(* IEC 61131-3 sources: platform/iec61131/st/osoST/examples, 8 files *)

(* ---- array.st ---- *)
VAR_GLOBAL
  a : ARRAY[0..4] OF DINT;
  i : DINT := 0;
  sum : DINT := 0;
END_VAR

PROCEDURE main()
  FOR i := 0 TO 4 DO
    a[i] := i * 10;
  END_FOR;
  sum := 0;
  FOR i := 0 TO 4 DO
    sum := sum + a[i];
  END_FOR;
  debug(sum);
  debug(a[2]);
END_PROCEDURE

(* ---- array_real.st ---- *)
VAR_GLOBAL
  r : ARRAY[1..3] OF REAL;
  s : REAL := 0.0;
END_VAR

PROCEDURE main()
  r[1] := 1.5;
  r[2] := r[1] * 2.0;
  r[3] := r[2] + r[1];
  s := r[1] + r[2] + r[3];
  debug(s);
  debug(r[3]);
END_PROCEDURE

(* ---- blink.st ---- *)
(* ============================================================
   osoLogic — IEC 61131-3 Structured Text example
   blink.st — LED blink using a counter and trap calls

   Copyright (C) 2026 Angel Miguel Zúñiga Schmemund <miguel@ibercomp.com>
                 Ibercomp SL, Roig Borrell SL

   Part of the osoLogic open-source PLC project — osologic.org
   SPDX-License-Identifier: AGPL-3.0-or-later

   Description / Descripción:
     Toggle a GPIO output every N scan cycles.
     Alterna una salida GPIO cada N ciclos de scan.

   Traps used / Traps utilizados:
     gpio_write(pin, value)  — trap #10
     millis()                — trap #12  (returns I32 milliseconds)
   ============================================================ *)

(* Hardware traps — link to hardware_linux.c or hardware_bare.c
   Traps de hardware — enlazar con hardware_linux.c o hardware_bare.c *)
TRAP gpio_write(pin : DINT; value : DINT) TRAP #10;
TRAP gpio_read(pin : DINT) : DINT        TRAP #11;
TRAP millis() : DINT                     TRAP #12;

(* ── Global state / Estado global ──────────────────────── *)
VAR_GLOBAL
  led_state    : BOOL  := FALSE;
  last_toggle  : DINT  := 0;
END_VAR

(* ── Constants / Constantes ─────────────────────────────── *)
VAR_GLOBAL
  LED_PIN      : DINT  := 0;   (* GPIO pin number / Número de pin GPIO *)
  BLINK_MS     : DINT  := 500; (* Toggle interval ms / Intervalo de alternancia ms *)
END_VAR

(* ── Main scan procedure / Procedimiento principal de scan ─ *)
PROCEDURE main()
VAR
  now : DINT;
END_VAR
  now := millis();
  IF (now - last_toggle) >= BLINK_MS THEN
    led_state   := NOT led_state;
    last_toggle := now;
    gpio_write(LED_PIN, led_state ? 1 : 0);
  END_IF;
END_PROCEDURE

(* ---- cast.st ---- *)
VAR_GLOBAL
  i : DINT := 7;
  x : REAL := 0.0;
  y : REAL := 0.0;
  z : DINT := 0;
END_VAR

PROCEDURE main()
  x := i * 2.5;
  y := TO_REAL(i) + 0.5;
  z := REAL_TO_INT(x);
  debug(x);
  debug(y);
  debug(z);
END_PROCEDURE

(* ---- counter.st ---- *)
(* ============================================================
   osoLogic — IEC 61131-3 Structured Text example
   counter.st — Up/down counter with debug output

   Copyright (C) 2026 Angel Miguel Zúñiga Schmemund <miguel@ibercomp.com>
                 Ibercomp SL, Roig Borrell SL

   Part of the osoLogic open-source PLC project — osologic.org
   SPDX-License-Identifier: AGPL-3.0-or-later

   Description / Descripción:
     Simple up counter incremented each scan cycle.
     Demonstrates: global variables, IF, debug output.
     Contador ascendente incrementado cada ciclo de scan.
     Demuestra: variables globales, IF, salida debug.
   ============================================================ *)

VAR_GLOBAL
  count    : DINT  := 0;
  max_val  : DINT  := 100;
  overflow : BOOL  := FALSE;
END_VAR

PROCEDURE main()
  count := count + 1;
  IF count >= max_val THEN
    count    := 0;
    overflow := TRUE;
    debug("Counter overflow / Desbordamiento del contador");
  ELSE
    overflow := FALSE;
  END_IF;
  debug(count);
END_PROCEDURE

(* ---- pid.st ---- *)
(* ============================================================
   osoLogic — IEC 61131-3 Structured Text example
   pid.st — Simple discrete PID controller

   Copyright (C) 2026 Angel Miguel Zúñiga Schmemund <miguel@ibercomp.com>
                 Ibercomp SL, Roig Borrell SL

   Part of the osoLogic open-source PLC project — osologic.org
   SPDX-License-Identifier: AGPL-3.0-or-later

   Description / Descripción:
     Position-form discrete PID (P + I + D terms).
     The scan cycle in osoruntime.c calls main() at a fixed period.
     Call pid_update() from your main procedure, passing the current
     process value and setpoint. Returns control output clamped to
     [out_min, out_max].

     PID discreto en forma posición (términos P + I + D).
     El ciclo de scan en osoruntime.c llama a main() a periodo fijo.
     Llame a pid_update() desde su procedimiento principal, pasando
     el valor de proceso actual y el setpoint. Devuelve la salida de
     control limitada a [out_min, out_max].

   Usage / Uso:
     output := pid_update(process_value, setpoint);
   ============================================================ *)

(* PID tuning parameters / Parámetros de sintonía PID *)
VAR_GLOBAL
  pid_kp      : REAL := 1.0;   (* Proportional gain / Ganancia proporcional *)
  pid_ki      : REAL := 0.1;   (* Integral gain     / Ganancia integral     *)
  pid_kd      : REAL := 0.05;  (* Derivative gain   / Ganancia derivativa   *)
  pid_out_min : REAL := -100.0;
  pid_out_max : REAL :=  100.0;
END_VAR

(* Internal state — do NOT modify from outside *)
(* Estado interno — NO modificar desde fuera   *)
VAR_GLOBAL
  _pid_integral : REAL := 0.0;
  _pid_prev_err : REAL := 0.0;
END_VAR

(* ── PID update function / Función de actualización PID ──── *)
FUNCTION pid_update : REAL
VAR_INPUT
  pv       : REAL;   (* Process value / Valor de proceso *)
  setpoint : REAL;   (* Desired value / Valor deseado    *)
END_VAR
VAR
  err    : REAL;
  p_term : REAL;
  d_term : REAL;
  output : REAL;
END_VAR
  err    := setpoint - pv;

  (* Proportional / Proporcional *)
  p_term := pid_kp * err;

  (* Integral with anti-windup clamp / Integral con límite anti-windup *)
  _pid_integral := _pid_integral + pid_ki * err;
  IF _pid_integral > pid_out_max THEN
    _pid_integral := pid_out_max;
  ELSIF _pid_integral < pid_out_min THEN
    _pid_integral := pid_out_min;
  END_IF;

  (* Derivative / Derivativo *)
  d_term := pid_kd * (err - _pid_prev_err);
  _pid_prev_err := err;

  (* Sum and clamp output / Suma y limitación de salida *)
  output := p_term + _pid_integral + d_term;
  IF output > pid_out_max THEN
    output := pid_out_max;
  ELSIF output < pid_out_min THEN
    output := pid_out_min;
  END_IF;

  pid_update := output;
END_FUNCTION

(* ── Demo main procedure / Procedimiento principal demo ──── *)
VAR_GLOBAL
  process_temp : REAL := 20.0;   (* Simulated sensor   / Sensor simulado   *)
  heater_out   : REAL := 0.0;    (* Heater power %     / Potencia calefactor % *)
END_VAR

PROCEDURE main()
VAR
  sp : REAL;
END_VAR
  sp          := 60.0;   (* Target temperature / Temperatura objetivo *)
  heater_out  := pid_update(process_temp, sp);
  (* Simulate plant response / Simular respuesta de planta *)
  process_temp := process_temp + 0.01 * heater_out - 0.005 * (process_temp - 20.0);
  debug(process_temp, heater_out);
END_PROCEDURE

(* ---- string.st ---- *)
VAR_GLOBAL
  msg : STRING := 'hello';
END_VAR

PROCEDURE main()
  debug(msg);
  debug('world');
END_PROCEDURE

(* ---- string_compare.st ---- *)
VAR_GLOBAL
  msg : STRING := 'on';
  matched : DINT := 0;
  other : DINT := 0;
END_VAR

PROCEDURE main()
  IF msg = 'on' THEN
    matched := 1;
  END_IF;
  IF msg = 'off' THEN
    other := 1;
  END_IF;
  debug(matched);
  debug(other);
END_PROCEDURE
